{attribute 'qualified_only'}
//{attribute 'strict'}
{attribute 'to_string'}
TYPE E_MESSAGE_STATE :
(
	MSG_STATE_NULL,
  MSG_STATE_INIT    := 10,
  MSG_STATE_IDLE    := 30,
  MSG_STATE_WRITE   := 50
)UINT;
END_TYPE

(* stored: Version 1.1.0.1, ProductVersion 3.1.4026.18
   DUT E_MESSAGE_STATE: Id {4aa5f62f-5886-4f20-946d-76e30a266395} *)
